// TIA Portal V17 export
// export: Created 2025-03-05T08:01:14.9739304Z, ExportSetting WithDefaults, DisplayName Totally Integrated Automation Portal, DisplayVersion V17 Update 8, DisplayName TIA Portal Openness, DisplayVersion V17 Update 8, DisplayName TIA Portal Version Control Interface, DisplayVersion V17, DisplayName SINAMICS Startdrive Advanced, DisplayVersion V17 SP2, DisplayName SINAMICS Startdrive G110M, G120, G120C, G120D, G120P, G115D, DisplayVersion V17 SP2, DisplayName SINAMICS Startdrive G130, G150, S120, S150, SINAMICS MV, S210, DisplayVersion V17 SP2, DisplayName STEP 7 Professional, DisplayVersion V17 Update 8, DisplayName SINUMERIK ONE STEP 7 Toolbox, DisplayVersion V17 Update 12, DisplayName SINUMERIK 840D sl STEP 7 Toolbox, DisplayVersion V17 Update 12, DisplayName STEP 7 Safety, DisplayVersion V17 Update 6, DisplayName WinCC Advanced, DisplayVersion V17 Update 8
FUNCTION "FC6500_CYLINDERS" : Void   // FC6500, LAD
{ S7_Optimized_Access := 'FALSE' }
AUTHOR : ETXETAR
VERSION : 1.0
// stored: AutoNumber false, IsIECCheckEnabled false, SetENOAutomatically false, UDAEnableTagReadback false
BEGIN

REGION Network 1: FC6600_UNIT_01_UP_SEALING_STRUCTURE
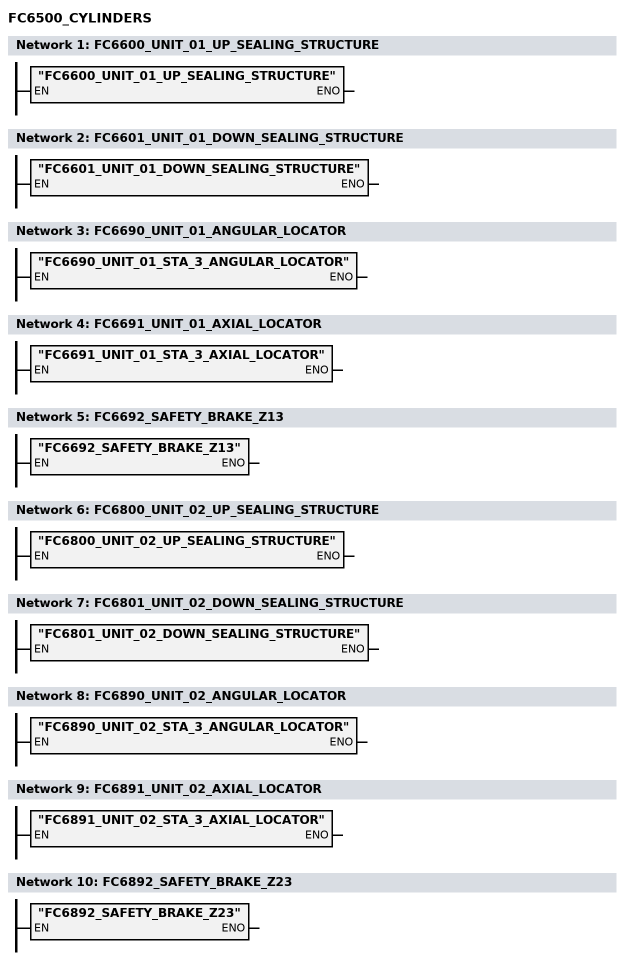
   RUNG wire#powerrail
      "FC6600_UNIT_01_UP_SEALING_STRUCTURE"()
   END_RUNG
   // the same network as SCL:
   "FC6600_UNIT_01_UP_SEALING_STRUCTURE"();
END_REGION

REGION Network 2: FC6601_UNIT_01_DOWN_SEALING_STRUCTURE
   RUNG wire#powerrail
      "FC6601_UNIT_01_DOWN_SEALING_STRUCTURE"()
   END_RUNG
   // the same network as SCL:
   "FC6601_UNIT_01_DOWN_SEALING_STRUCTURE"();
END_REGION

REGION Network 3: FC6690_UNIT_01_ANGULAR_LOCATOR
   RUNG wire#powerrail
      "FC6690_UNIT_01_STA_3_ANGULAR_LOCATOR"()
   END_RUNG
   // the same network as SCL:
   "FC6690_UNIT_01_STA_3_ANGULAR_LOCATOR"();
END_REGION

REGION Network 4: FC6691_UNIT_01_AXIAL_LOCATOR
   RUNG wire#powerrail
      "FC6691_UNIT_01_STA_3_AXIAL_LOCATOR"()
   END_RUNG
   // the same network as SCL:
   "FC6691_UNIT_01_STA_3_AXIAL_LOCATOR"();
END_REGION

REGION Network 5: FC6692_SAFETY_BRAKE_Z13
   RUNG wire#powerrail
      "FC6692_SAFETY_BRAKE_Z13"()
   END_RUNG
   // the same network as SCL:
   "FC6692_SAFETY_BRAKE_Z13"();
END_REGION

REGION Network 6: FC6800_UNIT_02_UP_SEALING_STRUCTURE
   RUNG wire#powerrail
      "FC6800_UNIT_02_UP_SEALING_STRUCTURE"()
   END_RUNG
   // the same network as SCL:
   "FC6800_UNIT_02_UP_SEALING_STRUCTURE"();
END_REGION

REGION Network 7: FC6801_UNIT_02_DOWN_SEALING_STRUCTURE
   RUNG wire#powerrail
      "FC6801_UNIT_02_DOWN_SEALING_STRUCTURE"()
   END_RUNG
   // the same network as SCL:
   "FC6801_UNIT_02_DOWN_SEALING_STRUCTURE"();
END_REGION

REGION Network 8: FC6890_UNIT_02_ANGULAR_LOCATOR
   RUNG wire#powerrail
      "FC6890_UNIT_02_STA_3_ANGULAR_LOCATOR"()
   END_RUNG
   // the same network as SCL:
   "FC6890_UNIT_02_STA_3_ANGULAR_LOCATOR"();
END_REGION

REGION Network 9: FC6891_UNIT_02_AXIAL_LOCATOR
   RUNG wire#powerrail
      "FC6891_UNIT_02_STA_3_AXIAL_LOCATOR"()
   END_RUNG
   // the same network as SCL:
   "FC6891_UNIT_02_STA_3_AXIAL_LOCATOR"();
END_REGION

REGION Network 10: FC6892_SAFETY_BRAKE_Z23
   RUNG wire#powerrail
      "FC6892_SAFETY_BRAKE_Z23"()
   END_RUNG
   // the same network as SCL:
   "FC6892_SAFETY_BRAKE_Z23"();
END_REGION
END_FUNCTION
